FUNCTION_BLOCK Mixer_Main (* Service Interface Function Block Type *)
  (* Standard: 61499-2 *)
  (* Version 1.0, 2023-08-25, ADMIN *)
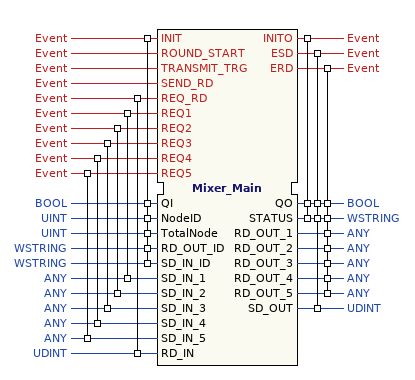
  EVENT_INPUT
    INIT WITH QI, NodeID, TotalNode, RD_OUT_ID, SD_IN_ID; (* Service Initialization *)
    ROUND_START;
    TRANSMIT_TRG;
    SEND_RD;
    REQ_RD WITH RD_IN;
    REQ1 WITH SD_IN_1;
    REQ2 WITH SD_IN_2;
    REQ3 WITH SD_IN_3;
    REQ4 WITH SD_IN_4;
    REQ5 WITH SD_IN_5;
  END_EVENT
  EVENT_OUTPUT
    INITO WITH QO, STATUS; (* Initialization Confirm *)
    ESD WITH QO, STATUS, SD_OUT; (* Confirmation of Requested Service *)
    ERD WITH RD_OUT_1, QO, STATUS, RD_OUT_2, RD_OUT_3, RD_OUT_4, RD_OUT_5;
  END_EVENT
  VAR_INPUT
    QI : BOOL; (* Event Input Qualifier *)
    NodeID : UINT; (* Current Node ID *)
    TotalNode : UINT; (* Total Node in System *)
    RD_OUT_ID : WSTRING;
    SD_IN_ID : WSTRING;
    SD_IN_1 : ANY;
    SD_IN_2 : ANY;
    SD_IN_3 : ANY;
    SD_IN_4 : ANY;
    SD_IN_5 : ANY;
    RD_IN : UDINT; (* Data from Network *)
  END_VAR
  VAR_OUTPUT
    QO : BOOL; (* Event Output Qualifier *)
    STATUS : WSTRING; (* Service Status *)
    RD_OUT_1 : ANY;
    RD_OUT_2 : ANY;
    RD_OUT_3 : ANY;
    RD_OUT_4 : ANY;
    RD_OUT_5 : ANY;
    SD_OUT : UDINT; (* Send Data to Network *)
  END_VAR
  (* Service APPLICATION/RESOURCE: Service Interface Function Block Type *)
END_FUNCTION_BLOCK
